{attribute 'qualified_only'}
{attribute 'to_string'}
TYPE E_DGPDState :
(
		UNKNOWN:=0,
        OUT,
        TARGET1A,
        TARGET1B,
        TARGET1C,
        TARGET1D,
        TARGET2,
        TARGET3,
        TARGET4,
        TARGET5,
        TARGET6
)UINT;
END_TYPE

(* stored: Version 1.1.0.1
   DUT E_DGPDState: Id {018f8515-71cb-4f89-95db-5b7ba67f56e9} *)
